(* IEC 61131-3 sources: JaccoSigma/tempclass/Class/RoundDown, 1 file *)

(* ---- RoundDown.st ---- *)
(*!
<Class
	Name               = "RoundDown"
	Revision           = "0.0"
	RealtimeTask       = "false"
	CyclicTask         = "false"
	BackgroundTask     = "false"
	Sigmatek           = "false"
	OSInterface        = "false"
	HighPriority       = "false"
	Automatic          = "false"
	UpdateMode         = "Prescan"
	SharedCommandTable = "true"
	Objectsize         = "(1170,240)">
	<Channels>
		<Server Name="DintOUT" Visualized="false" Initialize="false" WriteProtected="true" Retentive="false"/>
		<Server Name="RealIN" Visualized="false" Initialize="false" WriteProtected="false" Retentive="false"/>
	</Channels>
</Class>
*)
RoundDown : CLASS
  //Servers:
	RealIN 	: SvrChCmd_REAL;
	DintOUT 	: SvrCh_DINT;
  //Clients:
  //Variables:
		TempReal 	: REAL;
		TempDint 	: DINT;
  //Functions:

	FUNCTION VIRTUAL GLOBAL RealIN::Write
		VAR_INPUT
			input (EAX) 	: REAL;
		END_VAR
		VAR_OUTPUT
			result (EAX) 	: REAL;
		END_VAR;
  //Tables:
	FUNCTION @STD
		VAR_OUTPUT
			ret_code	: CONFSTATES;
		END_VAR;
	FUNCTION GLOBAL TAB @CT_;
END_CLASS;

FUNCTION VIRTUAL GLOBAL RoundDown::RealIN::Write
	VAR_INPUT
		input (EAX) 	: REAL;
	END_VAR
	VAR_OUTPUT
		result (EAX) 	: REAL;
	END_VAR

	RealIN := input;

  TempReal := (RealIN-0.5);
  DintOUT := to_dint(TempReal);

	result := RealIN;

END_FUNCTION
